FUNCTION_BLOCK Request_Manager (* Composite Function Block Type *)
  (* Standard: 61499-2 *)
  (* Version 0.0, 9/24/2026, macie, Schneider Electric, template *)
  PACKAGE Main;
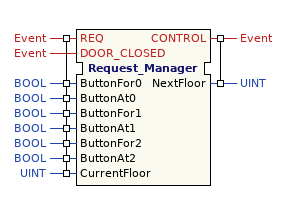
  EVENT_INPUT
    REQ WITH ButtonFor0, ButtonAt0, ButtonFor1, ButtonAt1, ButtonFor2, ButtonAt2, CurrentFloor; (* Normal Execution Request *)
    DOOR_CLOSED;
  END_EVENT
  EVENT_OUTPUT
    CONTROL WITH NextFloor; (* Execution Confirmation *)
  END_EVENT
  VAR_INPUT
    ButtonFor0 : BOOL; (* Input event qualifier *)
    ButtonAt0 : BOOL;
    ButtonFor1 : BOOL;
    ButtonAt1 : BOOL;
    ButtonFor2 : BOOL;
    ButtonAt2 : BOOL;
    CurrentFloor : UINT;
  END_VAR
  VAR_OUTPUT
    NextFloor : UINT; (* Output event qualifier *)
  END_VAR
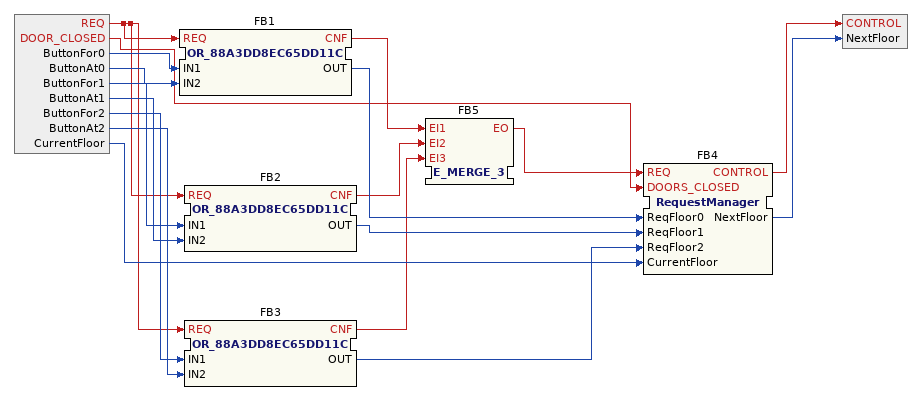
  FBS
    FB1 : OR_88A3DD8EC65DD11C; {SET_ATTRIBUTE(Configuration.GenericFBType.InterfaceParams, Runtime.Standard#CNT:=2;OUT:BOOL)}
    FB2 : OR_88A3DD8EC65DD11C; {SET_ATTRIBUTE(Configuration.GenericFBType.InterfaceParams, Runtime.Standard#CNT:=2;OUT:BOOL)}
    FB3 : OR_88A3DD8EC65DD11C; {SET_ATTRIBUTE(Configuration.GenericFBType.InterfaceParams, Runtime.Standard#CNT:=2;OUT:BOOL)}
    FB4 : RequestManager;
    FB5 : E_MERGE_3;
  END_FBS
  EVENT_CONNECTIONS
    REQ TO FB1.REQ;
    REQ TO FB2.REQ;
    REQ TO FB3.REQ;
    FB1.CNF TO FB5.EI1;
    FB2.CNF TO FB5.EI2;
    FB3.CNF TO FB5.EI3;
    FB5.EO TO FB4.REQ;
    FB4.CONTROL TO CONTROL;
    DOOR_CLOSED TO FB4.DOORS_CLOSED;
  END_CONNECTIONS
  DATA_CONNECTIONS
    ButtonFor0 TO FB1.IN1;
    ButtonAt0 TO FB1.IN2;
    ButtonFor1 TO FB2.IN1;
    ButtonAt1 TO FB2.IN2;
    ButtonFor2 TO FB3.IN1;
    ButtonAt2 TO FB3.IN2;
    FB1.OUT TO FB4.ReqFloor0;
    FB2.OUT TO FB4.ReqFloor1;
    FB3.OUT TO FB4.ReqFloor2;
    CurrentFloor TO FB4.CurrentFloor;
    FB4.NextFloor TO NextFloor;
  END_CONNECTIONS
END_FUNCTION_BLOCK
